PROGRAM MAIN
VAR
	bRunOnlyOnce : BOOL := FALSE;
END_VAR

IF NOT bRunOnlyOnce THEN
		ADSLOGSTR(msgCtrlMask := ADSLOG_MSGTYPE_ERROR OR ADSLOG_MSGTYPE_LOG, 
			msgFmtStr := 'Hello',
			strArg :='');
		bRunOnlyOnce := TRUE;
END_IF

END_PROGRAM

(* stored: Version 1.1.0.1, ProductVersion 3.1.4024.12
   POU MAIN: Id {c05b0674-bccf-482e-b624-f9e009c1cb09}, SpecialFunc None *)
